FUNCTION DebugLen : UDINT

DebugLen := _Debug.nDebugLen;

END_FUNCTION

(* stored: Version 1.1.0.1
   POU DebugLen: Id {c7995225-ddbc-416c-a07d-8450904a8422}, SpecialFunc None *)
